Universal Robots PolyScope program: g_to_a.urp

Program g_to_a (installation=string_planes directory=/programs/string_crossings createdIn=5.17.3 lastSavedIn=5.17.3 robotSerialNumber=20245501435)
Calibrated DH parameters: a=[0.000154, -0.137004, -0.385524, -0.00002, 0.000092, 0]; d=[0.162441, 211.794786, -230.585024, 18.923638, 0.099786, 0.09951]; alpha=[1.569493, -0.001902, 0.003874, 1.570111, -1.570167, 0]; deltaTheta=[0, -1.242934, 1.056292, 0.186646, 0.000002, 0.000001]
InitVariablesNode
Robot Program (runOnlyOnce=false)
  bow_section := -1
  If bow_section≟-1
    MoveJ speed 60 deg/s, acceleration 80 deg/s^2 (useActiveTCP=true) feature=Base
      Waypoint Waypoint_2 (Relative): relativeFromPosition TCP in base x=333.304 y=655.506 z=103.679 mm, rx=-1.6491 ry=-1.7982 rz=0.6657 rad; joints [-132.462, -27.759, 71.843, -100.48, -56.044, -147.727] deg; TCP offset x=28.21 y=-96.107 z=-99.69 mm, rx=0 ry=0 rz=0 rad; TCP in base x=277.25 y=734.024 z=156.888 mm, rx=1.739 ry=2.3104 rz=-1.1078 rad; joints [-126.649, -28.124, 54.73, -74.618, -91.963, -141.811] deg
  ElseIf bow_section≟0
    MoveJ speed 60 deg/s, acceleration 80 deg/s^2 (useActiveTCP=true) feature=Base
      Waypoint Waypoint_1 (Relative): relativeFromPosition TCP in base x=267.753 y=455.828 z=63.352 mm, rx=-1.6064 ry=-1.9107 rz=0.8701 rad; joints [-141.613, -39.193, 108.913, -115.288, -70.779, -159.12] deg; TCP in base x=327.364 y=541.729 z=231.867 mm, rx=1.6818 ry=2.3248 rz=-1.1114 rad; joints [-139.638, -50.32, 85.996, -84.695, -102.358, -153.079] deg
  Else 
    MoveJ speed 60 deg/s, acceleration 80 deg/s^2 (useActiveTCP=true) feature=Base
      Waypoint Waypoint_3 (Relative): relativeFromPosition TCP in base x=243.623 y=214.066 z=64.409 mm, rx=-1.5873 ry=-1.9212 rz=0.9621 rad; joints [-169.307, -44.602, 138.124, -133.879, -94.42, -177.776] deg; TCP in base x=374.975 y=359.143 z=303.031 mm, rx=1.6275 ry=2.3373 rz=-1.1145 rad; joints [-156.115, -66.366, 101.55, -88.735, -114.429, -168.117] deg
